PROGRAM FBDPOU
VAR
	// Start Button
	btnStart: BOOL;
	// Stop Button
	btnStop: BOOL;
	// Motor Starter Coil
	Coil: BOOL;
END_VAR

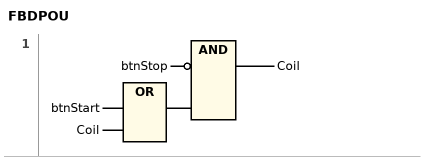
// NETWORK 1
Coil := NOT btnStop AND (btnStart OR Coil);

END_PROGRAM

(* stored: Version 1.1.0.1, ProductVersion 3.1.4024.15
   POU FBDPOU: Id {08b0a916-6ca2-4ddb-823c-8eca2cc5f3af}, SpecialFunc None *)
